FUNCTION_BLOCK FB_PizzaOven
VAR_INPUT
	
	bLoadPizza : BOOL;	// Put a pizza on the input side
	bRemovePizza : BOOL;	// Take pizza off output side

END_VAR
VAR_OUTPUT

	bBuzzer : BOOL;
	bLight : BOOL;

	iTotalPizzasCooked : UDINT;

END_VAR
VAR
	
	stCurrentTime : TIMESTRUCT;
	dtCurrentTime : DT;

	fbLoad_RTRIG : R_TRIG;
	fbRemove_RTRIG : R_TRIG;	

	stPizzaOnDeck : ST_PIZZA;	// Location of possible pizza
	stPizzaInOven : ST_PIZZA;
	stPizzaDone : ST_PIZZA;
	
	// timers
	fbMyTimer : TON;	// My timer... for stuff.

	iState : DINT;
	ILastState : DINT;
	sStateDesc : STRING;
	arrStateDescHistory : ARRAY[1..100] OF STRING;
	
	bStartButton: BOOL;
	arrPizzaHistory: BYTE;
	TIMESTR: STRING(INT#4);
END_VAR
VAR CONSTANT
	stNULL_PIZZA : ST_PIZZA;
END_VAR

dtCurrentTime := SYSTEMTIME_TO_DT(stCurrentTime);

// If there is room
IF stPizzaOnDeck.bExist AND NOT stPizzaInOven.bExist THEN
	stPizzaInOven := stPizzaOnDeck;
	stPizzaOnDeck := stNULL_PIZZA;	// Remove pizza
END_IF

fbLoad_RTRIG(clk := bLoadPizza);
IF fbLoad_RTRIG.Q THEN
	stPizzaOnDeck.bExist := TRUE;
	stPizzaOnDeck.eType := 2;	// Olives
END_IF

fbRemove_RTRIG(clk := bRemovePizza);
IF fbRemove_RTRIG.Q THEN
	//F_FIFO_WRITE(cbData := SIZEOF(stPizzaDone), pData := ADR(stPizzaDone),
	//				cbBuffer := SIZEOF(arrPizzaHistory), pBuffer := ADR(arrPizzaHistory)
	//);	//It gives an error for arrPizzaHistory, I don't know how to fix it
	stPizzaDone := stNULL_PIZZA;
END_IF

CASE iState OF
	0:	// Wait for pizza in oven
		sStateDesc := 'Waiting on pizza now.';
		IF stPizzaInOven.bExist THEN
			stPizzaInOven.dtTimeEnteredOven := dtCurrentTime;
			iState := 10;
		END_IF
	10:	// We just got a pizza!
		sStateDesc := 'Baking that pizza now.';
		fbMyTimer(IN:=TRUE, PT:=T#3S);
		
		IF fbMyTimer.Q THEN
			fbMyTimer(IN:=FALSE);
			iState := 20;
		END_IF
	20:	// Can we move the pizza out of the oven? It's going to burn!
		IF NOT stPizzaDone.bExist THEN
			// Simulate conveyor
			stPizzaInOven.dtTimeExitedOven := dtCurrentTime;
			stPizzaDone := stPizzaInOven;
			stPizzaInOven := stNULL_PIZZA;
			bBuzzer := FALSE;
			iState := 30;
		ELSE
			bBuzzer := TRUE;
			sStateDesc := 'The pizza is burning!';
		END_IF
	30:	// Pizza just removed on output tray
		stPizzaInOven.tTimeInOven := stPizzaInOven.dtTimeExitedOven - stPizzaInOven.dtTimeEnteredOven;
		iTotalPizzasCooked := iTotalPizzasCooked + 1;
		iState := 0;	// Go wait for new pizza in oven!
ELSE
	sStateDesc := 'Invalid state!';
END_CASE

// Start state history

IF iLastState <> iState THEN
	// Do stuff here to log transitions...
	F_FIFO_WRITE(cbData := SIZEOF(sStateDesc), pData := ADR(sStateDesc),
					cbBuffer := SIZEOF(arrStateDescHistory), pBuffer := ADR(arrStateDescHistory)
	);
	// ^^ SIZEOF returns the count in bytes
	
	// Reset for next time
	iLastState := iState;
END_IF

END_FUNCTION_BLOCK

(* stored: Version 1.1.0.1, ProductVersion 3.1.4024.12
   POU FB_PizzaOven: Id {5c55f55f-47e0-45bd-aa5b-72804a871bfe}, SpecialFunc None *)
